{attribute 'qualified_only'}
VAR_GLOBAL
	IP			:STRING(MAX_STRING_LENGTH) := 'opc.tcp://169.254.240.2:4840';
	NameSpace	:STRING(MAX_STRING_LENGTH) := 'urn:BeckhoffAutomation:Ua:PLC1';
	
	SW		:SystemStatusWord;
	CW		:SystemControlWord;
END_VAR

(* stored: Version 1.1.0.1, ProductVersion 3.1.4024.12
   GVL GVL: Id {74ea964d-9a6c-4832-ba33-a0aebbba1e3b} *)
